// TIA Portal V16 export
// export: Created 2022-11-17T15:49:31.5042368Z, ExportSetting WithDefaults, DisplayName Totally Integrated Automation Portal, DisplayVersion V16 Update 6, DisplayName TIA Portal Version Control Interface, DisplayVersion V16 Update 2, DisplayName TIA Portal Openness, DisplayVersion V16 Update 6, DisplayName SINAMICS Startdrive Advanced, DisplayVersion V16 Update 5, DisplayName SINAMICS Startdrive G130, G150, S120, S150, SINAMICS MV, S210, DisplayVersion V16 Update 5, DisplayName SINAMICS Startdrive G110M, G120, G120C, G120D, G120P, G115D, DisplayVersion V16 Update 5, DisplayName STEP 7 Professional, DisplayVersion V16 Update 6, DisplayName STEP 7 Safety, DisplayVersion V16, DisplayName WinCC Advanced, DisplayVersion V16 Update 6
FUNCTION "FC102_EncoderCheck" : Void   // FC102, LAD
{ S7_Optimized_Access := 'FALSE' }
AUTHOR : AetnaG
VERSION : 0.0
// stored: AutoNumber false, IsIECCheckEnabled false, SetENOAutomatically false, UDAEnableTagReadback false
   VAR_INPUT
      MotorFwd : Bool;
      MotorBkw : Bool;
      AxisReset : Bool;
      EncValue : DInt;
      EncControl : DInt;
      Preset1 : Int;
      Preset2 : Int;
   END_VAR
   VAR_OUTPUT
      Alarm1 : Bool;
      Alarm2 : Bool;
   END_VAR
   VAR_IN_OUT
      LastEncValue : DInt;
      CounterDelay : Int;
      DelayDone : Bool;
      OneShootRise : Bool;
   END_VAR
   VAR_TEMP
      EncDifference : DInt;
      EncControlOpp : DInt;
      CounterReset : Bool;
   END_VAR
   VAR_TEMP   // added for the SCL form of the ladder/FBD networks
      _w1 : Bool;
   END_VAR
BEGIN

REGION Network 1
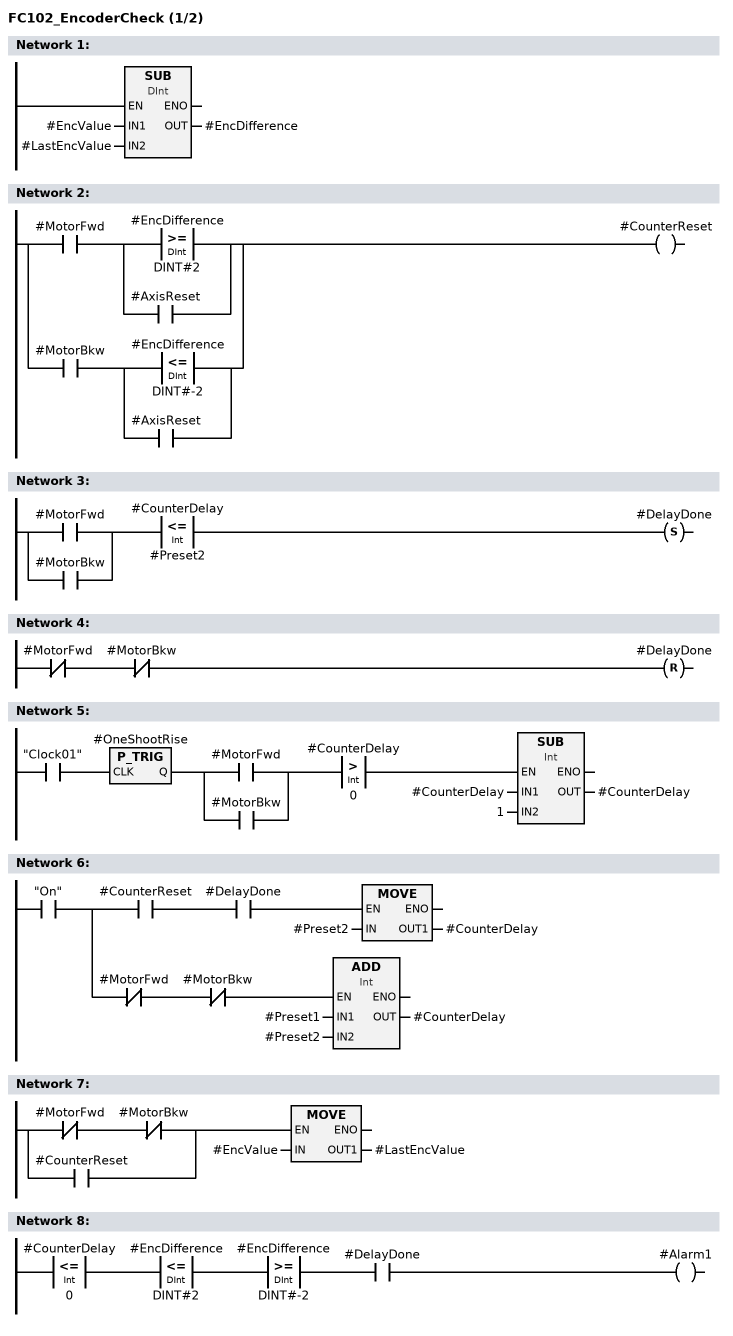
   RUNG wire#powerrail
      { S7_Templates := "SrcType := DInt"; S7_GenerateENO := "TRUE" } Sub(in1 := #EncValue, in2 := #LastEncValue, out => #EncDifference)
   END_RUNG
   // the same network as SCL:
   #EncDifference := #EncValue - #LastEncValue;
END_REGION

REGION Network 2
   RUNG wire#powerrail
      Contact( #MotorFwd )
      wire#w1
      { S7_Templates := "SrcType := DInt" } GE_Contact(in1 := #EncDifference, in2 := DINT#2)
      wire#w2
      Coil( #CounterReset )
   END_RUNG
   RUNG wire#w1
      Contact( #AxisReset )
   END_RUNG wire#w2
   RUNG wire#powerrail
      Contact( #MotorBkw )
      wire#w3
      { S7_Templates := "SrcType := DInt" } LE_Contact(in1 := #EncDifference, in2 := DINT#-2)
   END_RUNG wire#w2
   RUNG wire#w3
      Contact( #AxisReset )
   END_RUNG wire#w2
   // the same network as SCL:
   #CounterReset := (#MotorFwd AND ((#EncDifference >= DINT#2) OR #AxisReset)) OR (#MotorBkw AND ((#EncDifference <= DINT#-2) OR #AxisReset));
END_REGION

REGION Network 3
   RUNG wire#powerrail
      Contact( #MotorFwd )
      wire#w1
      { S7_Templates := "SrcType := Int" } LE_Contact(in1 := #CounterDelay, in2 := #Preset2)
      S_Coil( #DelayDone )
   END_RUNG
   RUNG wire#powerrail
      Contact( #MotorBkw )
   END_RUNG wire#w1
   // the same network as SCL:
   IF (#MotorFwd OR #MotorBkw) AND (#CounterDelay <= #Preset2) THEN #DelayDone := TRUE; END_IF;
END_REGION

REGION Network 4
   RUNG wire#powerrail
      I_Contact( #MotorFwd )
      I_Contact( #MotorBkw )
      R_Coil( #DelayDone )
   END_RUNG
   // the same network as SCL:
   IF NOT #MotorFwd AND NOT #MotorBkw THEN #DelayDone := FALSE; END_IF;
END_REGION

REGION Network 5
   RUNG wire#powerrail
      Contact( "Clock01" )
      P_Trig( #OneShootRise )
      wire#w1
      Contact( #MotorFwd )
      wire#w2
      { S7_Templates := "SrcType := Int" } GT_Contact(in1 := #CounterDelay, in2 := 0)
      { S7_Templates := "SrcType := Int"; S7_GenerateENO := "TRUE" } Sub(in1 := #CounterDelay, in2 := 1, out => #CounterDelay)
   END_RUNG
   RUNG wire#w1
      Contact( #MotorBkw )
   END_RUNG wire#w2
   // the same network as SCL:
   #_w1 := "Clock01" AND NOT #OneShootRise;   // rising edge
   #OneShootRise := "Clock01";
   IF #_w1 AND (#MotorFwd OR #MotorBkw) AND (#CounterDelay > 0) THEN
       #CounterDelay := #CounterDelay - 1;
   END_IF;
END_REGION

REGION Network 6
   RUNG wire#powerrail
      Contact( "On" )
      wire#w1
      Contact( #CounterReset )
      Contact( #DelayDone )
      { S7_GenerateENO := "TRUE" } Move(in := #Preset2, out1 => #CounterDelay)
   END_RUNG
   RUNG wire#w1
      I_Contact( #MotorFwd )
      I_Contact( #MotorBkw )
      { S7_Templates := "SrcType := Int"; S7_GenerateENO := "TRUE" } Add(in1 := #Preset1, in2 := #Preset2, out => #CounterDelay)
   END_RUNG
   // the same network as SCL:
   IF "On" AND #CounterReset AND #DelayDone THEN #CounterDelay := #Preset2; END_IF;
   IF "On" AND NOT #MotorFwd AND NOT #MotorBkw THEN #CounterDelay := #Preset1 + #Preset2; END_IF;
END_REGION

REGION Network 7
   RUNG wire#powerrail
      I_Contact( #MotorFwd )
      I_Contact( #MotorBkw )
      wire#w1
      { S7_GenerateENO := "TRUE" } Move(in := #EncValue, out1 => #LastEncValue)
   END_RUNG
   RUNG wire#powerrail
      Contact( #CounterReset )
   END_RUNG wire#w1
   // the same network as SCL:
   IF (NOT #MotorFwd AND NOT #MotorBkw) OR #CounterReset THEN #LastEncValue := #EncValue; END_IF;
END_REGION

REGION Network 8
   RUNG wire#powerrail
      { S7_Templates := "SrcType := Int" } LE_Contact(in1 := #CounterDelay, in2 := 0)
      { S7_Templates := "SrcType := DInt" } LE_Contact(in1 := #EncDifference, in2 := DINT#2)
      { S7_Templates := "SrcType := DInt" } GE_Contact(in1 := #EncDifference, in2 := DINT#-2)
      Contact( #DelayDone )
      Coil( #Alarm1 )
   END_RUNG
   // the same network as SCL:
   #Alarm1 := (#CounterDelay <= 0) AND (#EncDifference <= DINT#2) AND (#EncDifference >= DINT#-2) AND #DelayDone;
END_REGION

REGION Network 9
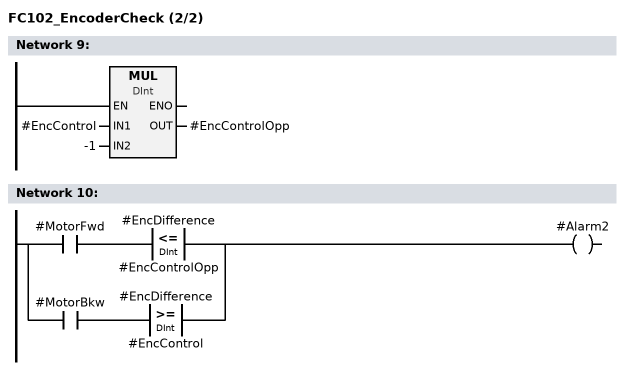
   RUNG wire#powerrail
      { S7_Templates := "SrcType := DInt"; S7_GenerateENO := "TRUE" } Mul(in1 := #EncControl, in2 := -1, out => #EncControlOpp)
   END_RUNG
   // the same network as SCL:
   #EncControlOpp := #EncControl * (-1);
END_REGION

REGION Network 10
   RUNG wire#powerrail
      Contact( #MotorFwd )
      { S7_Templates := "SrcType := DInt" } LE_Contact(in1 := #EncDifference, in2 := #EncControlOpp)
      wire#w1
      Coil( #Alarm2 )
   END_RUNG
   RUNG wire#powerrail
      Contact( #MotorBkw )
      { S7_Templates := "SrcType := DInt" } GE_Contact(in1 := #EncDifference, in2 := #EncControl)
   END_RUNG wire#w1
   // the same network as SCL:
   #Alarm2 := (#MotorFwd AND (#EncDifference <= #EncControlOpp)) OR (#MotorBkw AND (#EncDifference >= #EncControl));
END_REGION
END_FUNCTION
